// 40 Visualizations/IO_FB/Parameter/Parameter_DO/VIS_PARAMETER_TEMP_DO
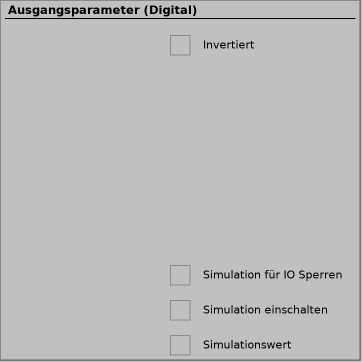
VISUALIZATION VIS_PARAMETER_TEMP_DO  // 362x362
VAR_INPUT
    ITF_DO_IN	:  	ITF_DO;
END_VAR
    RoundedRectangle (0,0 360x360)
    Label (5,0 350x20), "Ausgangsparameter (Digital)"
    Line (5,18) (355,18)
    Frame (170,35 20x20)
        shows CtaSysConfig.visBOOL(visfbBOOLIn := ITF_DO_IN.P_scfbDO_fbxInvert)
    Label (200,35 150x20), "Invertiert"
    Frame (170,335 20x20), invisible if: CtaSysConfig.fcGetEnumerationId(ITF_DO_IN.P_scfbIO_fbxSimulationLock) = 1
        shows CtaSysConfig.visBOOL(visfbBOOLIn := ITF_DO_IN.P_scfbDO_fbxSimulationValue)
    Label (200,335 150x20), "Simulationswert", invisible if: CtaSysConfig.fcGetEnumerationId(ITF_DO_IN.P_scfbIO_fbxSimulationLock) = 1
    Frame (170,265 20x20)
        shows CtaSysConfig.visBOOL(visfbBOOLIn := ITF_DO_IN.P_scfbIO_fbxSimulationLock)
    Label (200,300 150x20), "Simulation einschalten", invisible if: CtaSysConfig.fcGetEnumerationId(ITF_DO_IN.P_scfbIO_fbxSimulationLock) = 1
    Label (200,265 150x20), "Simulation für IO Sperren"
    Frame (170,300 20x20), invisible if: CtaSysConfig.fcGetEnumerationId(ITF_DO_IN.P_scfbIO_fbxSimulationLock) = 1
        shows CtaSysConfig.visBOOL(visfbBOOLIn := ITF_DO_IN.P_scfbIO_Simulation)
END_VISUALIZATION

// 40 Visualizations/IO_FB/DI/SimDI_Temp_Querry
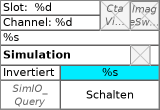
VISUALIZATION SimDI_Temp_Querry  // 160x110
VAR_INPUT
	ITF_DI : ITF_DI;
END_VAR
    Frame (0,0 160x110)
        shows SimDI_Temp(ITF_DI := ITF_DI)
END_VISUALIZATION

// 40 Visualizations/IO_FB/DO/SimDO_Temp_Querry
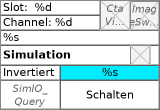
VISUALIZATION SimDO_Temp_Querry  // 160x110
VAR_INPUT	
	ITF_DO : ITF_DO;
END_VAR
    Frame (0,0 160x110)
        shows SimDO_Temp(ITF_DO := ITF_DO)
END_VISUALIZATION

// 40 Visualizations/IO_MANAGER/DEVICE/VIS_DEVICE_QUERY
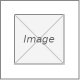
VISUALIZATION VIS_DEVICE_QUERY  // 80x80
VAR_INPUT
	ITF_IO_DEVICE_IN	:	ITF_IO_DEVICE;	
END_VAR
VAR
    fbDialog    	:   VU.FbOpenDialogExtended;
END_VAR
    Image (14,14 50x50), colour toggle: ITF_IO_DEVICE_IN.ERROR, input disabled if: ITF_IO_DEVICE_IN.proVISU_DIA_NAME = ''
        p84334746: ITF_IO_DEVICE_IN.IMAGE
        OnMouseClick: execute {
            ITF_IO_DEVICE_IN.RELOAD_ARRAY(TRUE,FALSE,FALSE);
            fbDialog(itfClientFilter            := VU.Globals.CurrentClient,
                     xExecute                   := FALSE,
            		 xModal						:= FALSE,
                     sDialogName                := ITF_IO_DEVICE_IN.proVISU_DIA_NAME,
                     pbyDialogInterfaceData     := ADR(ITF_IO_DEVICE_IN),
                     udiDialogInterfaceDataSize := SIZEOF(ITF_IO_DEVICE_IN));
            fbDialog(itfClientFilter            := VU.Globals.CurrentClient,
                     xExecute                   := TRUE,
            		 xModal						:= FALSE,
                     sDialogName                := ITF_IO_DEVICE_IN.proVISU_DIA_NAME,
                     pbyDialogInterfaceData     := ADR(ITF_IO_DEVICE_IN),
                     udiDialogInterfaceDataSize := SIZEOF(ITF_IO_DEVICE_IN));
        }
    Textfield (0,0 20x15), "%d", text variable: ITF_IO_DEVICE_IN.DEV_NR
    Textfield (0,65 80x15), "%s", text variable: ITF_IO_DEVICE_IN.proGetBMK
END_VISUALIZATION

// 40 Visualizations/IO_MANAGER/DIA_IO_DEVICES
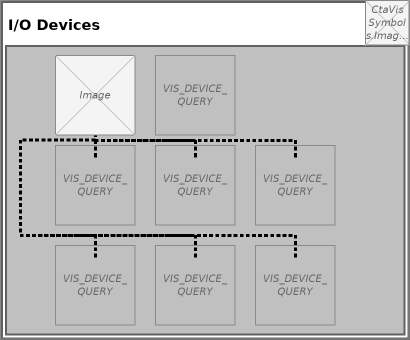
VISUALIZATION DIA_IO_DEVICES  // 410x340
VAR_INPUT
	ITF_IO_MANAGER_IN	:	ITF_IO_MANAGER;	
END_VAR
    RoundedRectangle (0,0 410x340)
    Frame (5,45 400x290), invisible if: NOT __QUERYINTERFACE(ITF_IO_MANAGER_IN,ITF_IO_MANAGER_IN)
        shows VIS_IO_DEVICES(ITF_IO_MANAGER_IN := ITF_IO_MANAGER_IN)
    Image (365,0 45x45), image: CtaVisSymbols.ImagePool.close_solo_black
        OnMouseClick:  Dialog=Current Dialog, Result=None, NumpadKeypadSet=True
    Label (5,5 150x40), "I/O Devices"
    InvisibleInput (5,2 360x40)
END_VISUALIZATION

// 40 Visualizations/IO_MANAGER/NETZWERK/VIS_IO_DEVICES
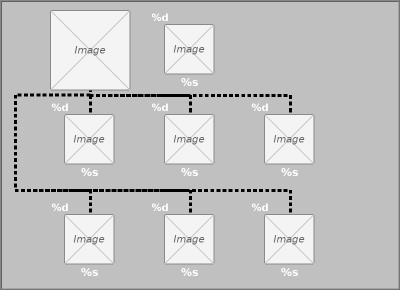
VISUALIZATION VIS_IO_DEVICES  // 400x290
VAR_INPUT
	ITF_IO_MANAGER_IN	:	ITF_IO_MANAGER;	
END_VAR
    Frame (0,0 400x290), invisible if: NOT __QUERYINTERFACE(ITF_IO_MANAGER_IN,ITF_IO_MANAGER_IN)
        shows VIS_IO_DEVICES_NETWORK(ITF_IO_MANAGER_IN := ITF_IO_MANAGER_IN, AY_ITF_DEVICE_VIS := ITF_IO_MANAGER_IN.AY_ITF_DEVICE_VIS)
END_VISUALIZATION

// 40 Visualizations/IO_MANAGER/NETZWERK/VIS_IO_DEVICES_NETWORK
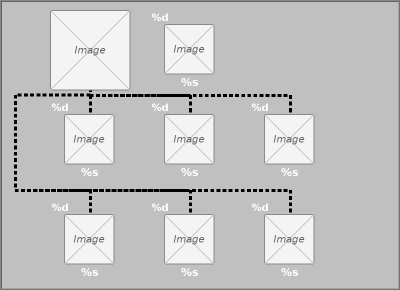
VISUALIZATION VIS_IO_DEVICES_NETWORK  // 400x290
VAR_INPUT
	ITF_IO_MANAGER_IN	:	ITF_IO_MANAGER;	
	AY_ITF_DEVICE_VIS 	: 	ARRAY[0..6] OF ITF_IO_DEVICE;
END_VAR
    RoundedRectangle (0,0 400x290)
    Frame (50,100 80x80)
        shows VIS_DEVICE(ITF_IO_DEVICE_IN := AY_ITF_DEVICE_VIS[1])
    Frame (150,100 80x80)
        shows VIS_DEVICE(ITF_IO_DEVICE_IN := AY_ITF_DEVICE_VIS[2])
    Frame (250,100 80x80)
        shows VIS_DEVICE(ITF_IO_DEVICE_IN := AY_ITF_DEVICE_VIS[3])
    Frame (50,200 80x80)
        shows VIS_DEVICE(ITF_IO_DEVICE_IN := AY_ITF_DEVICE_VIS[4])
    Frame (150,200 80x80)
        shows VIS_DEVICE(ITF_IO_DEVICE_IN := AY_ITF_DEVICE_VIS[5])
    Frame (250,200 80x80)
        shows VIS_DEVICE(ITF_IO_DEVICE_IN := AY_ITF_DEVICE_VIS[6])
    Frame (150,10 80x80)
        shows VIS_DEVICE(ITF_IO_DEVICE_IN := AY_ITF_DEVICE_VIS[0])
    Polyline (90,95) (15,95) (15,190) (90,190) (90,215), invisible if: AY_ITF_DEVICE_VIS[4] = 0
    Polyline (90,95) (15,95) (15,190) (190,190) (190,215), invisible if: AY_ITF_DEVICE_VIS[5] = 0
    Polyline (90,95) (15,95) (15,190) (290,190) (290,215), invisible if: AY_ITF_DEVICE_VIS[6] = 0
    Polyline (90,80) (90,95) (90,95) (290,95) (290,115), invisible if: AY_ITF_DEVICE_VIS[3] = 0
    Polyline (90,80) (90,95) (90,95) (190,95) (190,115), invisible if: AY_ITF_DEVICE_VIS[2] = 0
    Polyline (90,80) (90,95) (90,95) (90,95) (90,115), invisible if: ITF_IO_MANAGER_IN.COUNT = 0 AND AY_ITF_DEVICE_VIS[0] = 0
    Image (50,10 80x80), invisible if: __QUERYINTERFACE(AY_ITF_DEVICE_VIS[0],AY_ITF_DEVICE_VIS[0])
        p84334746: ITF_IO_MANAGER_IN.IMAGE
END_VISUALIZATION

// 40 Visualizations/IO_FB/Simulation/DIA_IO_CONFIG
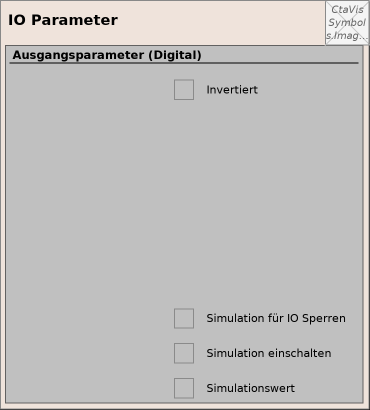
VISUALIZATION DIA_IO_CONFIG  // 370x410
VAR_INPUT
    ITF_IO_IN 	: 	ITF_IO;
END_VAR
    RoundedRectangle (0,0 370x410)
    Frame (5,45 360x360)
        shows VIS_IO_PARAMETER_BASE(ITF_IO_IN := ITF_IO_IN)
    Image (325,0 45x45), image: CtaVisSymbols.ImagePool.close_solo_black
        OnMouseClick:  Dialog=DIA_IO_CONFIG, Result=OK, NumpadKeypadSet=True
    Label (5,5 150x30), "IO Parameter"
    InvisibleInput (5,0 321x45)
END_VISUALIZATION

// 40 Visualizations/IO_TABLE/VIS_IO_TABLE
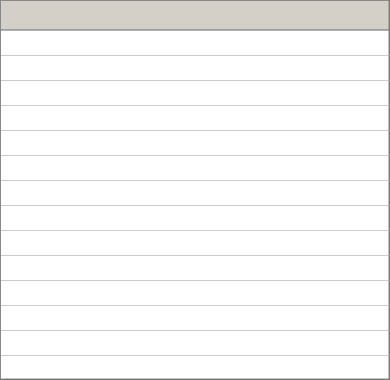
VISUALIZATION VIS_IO_TABLE  // 390x380
VAR_INPUT
	ITF_IO_SLOT_IN	:	ITF_IO_SLOT;	
END_VAR
VAR
	iMax			:	INT;
END_VAR
    Frame (0,0 390x380), invisible if: NOT __QUERYINTERFACE(ITF_IO_SLOT_IN,ITF_IO_SLOT_IN)
        shows VIS_IO_TABLE_QUERY(VIS_IO_TABLE := FC_VIS_IO_TABLE(ITF_IO_SLOT_IN := ITF_IO_SLOT_IN,iMax => iMax), iMax := iMax)
END_VISUALIZATION

// 40 Visualizations/IO_SLOT/VIS_IO_SLOT_IOS_ARRAY
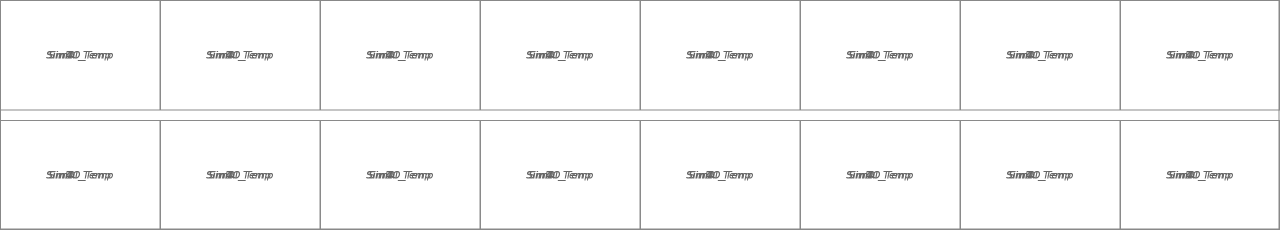
VISUALIZATION VIS_IO_SLOT_IOS_ARRAY  // 1280x230
VAR_INPUT
	AY_ITF_IO_VIS : ARRAY[1..16] OF ITF_IO;	
END_VAR
    Frame (0,0 160x110)
        shows Simulation(ITF_IO := AY_ITF_IO_VIS[1])
    Frame (160,0 160x110)
        shows Simulation(ITF_IO := AY_ITF_IO_VIS[2])
    Frame (320,0 160x110)
        shows Simulation(ITF_IO := AY_ITF_IO_VIS[3])
    Frame (480,0 160x110)
        shows Simulation(ITF_IO := AY_ITF_IO_VIS[4])
    Frame (640,0 160x110)
        shows Simulation(ITF_IO := AY_ITF_IO_VIS[5])
    Frame (800,0 160x110)
        shows Simulation(ITF_IO := AY_ITF_IO_VIS[6])
    Frame (960,0 160x110)
        shows Simulation(ITF_IO := AY_ITF_IO_VIS[7])
    Frame (1120,0 160x110)
        shows Simulation(ITF_IO := AY_ITF_IO_VIS[8])
    Frame (0,120 160x110)
        shows Simulation(ITF_IO := AY_ITF_IO_VIS[9])
    Frame (160,120 160x110)
        shows Simulation(ITF_IO := AY_ITF_IO_VIS[10])
    Frame (320,120 160x110)
        shows Simulation(ITF_IO := AY_ITF_IO_VIS[11])
    Frame (480,120 160x110)
        shows Simulation(ITF_IO := AY_ITF_IO_VIS[12])
    Frame (640,120 160x110)
        shows Simulation(ITF_IO := AY_ITF_IO_VIS[13])
    Frame (800,120 160x110)
        shows Simulation(ITF_IO := AY_ITF_IO_VIS[14])
    Frame (960,120 160x110)
        shows Simulation(ITF_IO := AY_ITF_IO_VIS[15])
    Frame (1120,120 160x110)
        shows Simulation(ITF_IO := AY_ITF_IO_VIS[16])
END_VISUALIZATION

// 40 Visualizations/IO_SLOT/VIS_IO_SLOT_IOS_QUERY
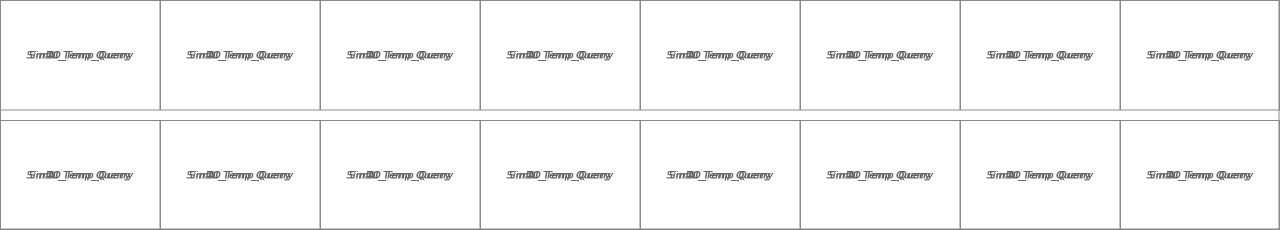
VISUALIZATION VIS_IO_SLOT_IOS_QUERY  // 1280x230
VAR_INPUT
	ITF_IO_SLOT_IN	:	ITF_IO_SLOT;	
END_VAR
    Frame (0,0 1280x230)
        shows VIS_IO_SLOT_IOS_ARRAY(AY_ITF_IO_VIS := ITF_IO_SLOT_IN.AY_ITF_IO_VIS)
END_VISUALIZATION

// 40 Visualizations/IO_SLOT/VIS_IO_SLOT_IOS
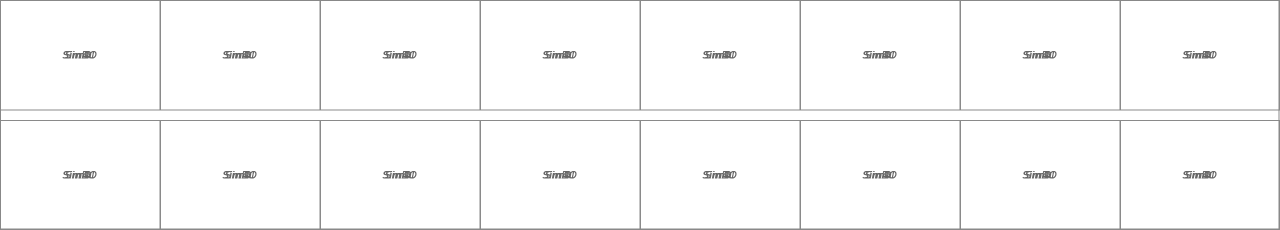
VISUALIZATION VIS_IO_SLOT_IOS  // 1280x230
VAR_INPUT
	ITF_IO_SLOT_IN	:	ITF_IO_SLOT;	
END_VAR
    Frame (0,0 1280x230), invisible if: NOT __QUERYINTERFACE(ITF_IO_SLOT_IN,ITF_IO_SLOT_IN)
        shows VIS_IO_SLOT_IOS_QUERY(ITF_IO_SLOT_IN := ITF_IO_SLOT_IN)
END_VISUALIZATION

// 40 Visualizations/IO_TABLE/VIS_IO_TABLE_QUERY
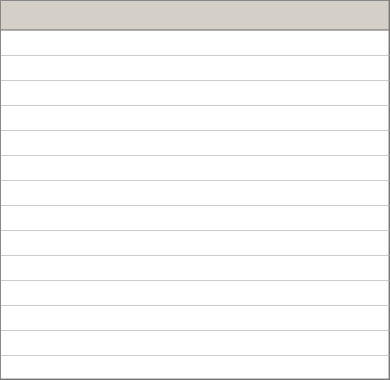
VISUALIZATION VIS_IO_TABLE_QUERY  // 390x380
VAR_INPUT
	VIS_IO_TABLE 	: ARRAY[1..18] OF ITF_IO_TABLE;
	iMax			: INT;
END_VAR
    Table (0,0 390x380), data array: VIS_IO_TABLE
        p1014161805: 18 - 1 + INT#1
        p1128707560: iMax
        p4242324053: FC_VIS_IO_TABLE(ITF_IO_SLOT_IN)[INDEX].proOkVisu
        p1739542657: FC_VIS_IO_TABLE(ITF_IO_SLOT_IN)[INDEX].proOK
        p516019884: FC_VIS_IO_TABLE(ITF_IO_SLOT_IN)[INDEX].proLogName
        p2243050616: FC_VIS_IO_TABLE(ITF_IO_SLOT_IN)[INDEX].proIsSimLocked
        p4088588272: FC_VIS_IO_TABLE(ITF_IO_SLOT_IN)[INDEX].proIsBOOL_IO
        p1757482276: FC_VIS_IO_TABLE(ITF_IO_SLOT_IN)[INDEX].PARENT
        p2192122294: FC_VIS_IO_TABLE(ITF_IO_SLOT_IN)[INDEX].proPhysikalValueVisu
        p400160035: FC_VIS_IO_TABLE(ITF_IO_SLOT_IN)[INDEX].ProSetInstancePathOnDynCreate
        p1265227338: FC_VIS_IO_TABLE(ITF_IO_SLOT_IN)[INDEX].proSimVisu
        p3726181087: FC_VIS_IO_TABLE(ITF_IO_SLOT_IN)[INDEX].SELF
        p3136911649: FC_VIS_IO_TABLE(ITF_IO_SLOT_IN)[INDEX].SELFPOINTER^
        p3854506369: VIS_IO_TABLE[INDEX].IO_NR
        p2170511999: VIS_IO_TABLE[INDEX].proPhysikalValueVisu
        p3723444502: VIS_IO_TABLE[INDEX].proSimVisu
        p1218418051: VIS_IO_TABLE[INDEX].SLOT_NR
        p2232123230: SLOT NR
        p511219082: IO NR
        p1755163831: IO TYPE
        p1791247317: VIS_IO_TABLE[INDEX].IO_TYPE
        p262371475: VIS_IO_TABLE[INDEX].proOkVisu
END_VISUALIZATION

// 40 Visualizations/IO_FB/IO/SimIO
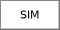
VISUALIZATION SimIO  // 60x30
VAR_INPUT	
	ITF_IO : ITF_IO;
END_VAR
VAR
	ITF_BOOL : CtaSysConfig.ITF_BOOL;
END_VAR
    Frame (0,0 60x30), invisible if: NOT __QUERYINTERFACE(ITF_IO.P_scfbIO_Simulation,ITF_BOOL), input disabled if: ITF_IO.proIsSimLocked
        shows SimIO_Temp(ITF_BOOL := ITF_BOOL)
END_VISUALIZATION

// 40 Visualizations/IO_FB/IO/SimIO_Query
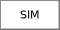
VISUALIZATION SimIO_Query  // 60x30
VAR_INPUT	
	ITF_BOOL : CtaSysConfig.ITF_BOOL;
END_VAR
    RoundedRectangle (0,0 60x30), "SIM", colour toggle: ITF_BOOL.proValue
        toggle ITF_BOOL.proValue
END_VISUALIZATION

// 40 Visualizations/IO_FB/DO/SimValue/SimDO_Value
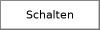
VISUALIZATION SimDO_Value  // 100x30
VAR_INPUT	
	ITF_DO : ITF_DO;
END_VAR
VAR
	ITF_BOOL : CtaSysConfig.ITF_BOOL;
END_VAR
    Frame (0,0 100x30), invisible if: NOT __QUERYINTERFACE(ITF_DO.P_scfbDO_fbxSimulationValue,ITF_BOOL), input disabled if: ITF_DO.proIsSimLocked
        shows SimDO_Value_Query(ITF_DO := ITF_DO, ITF_BOOL := ITF_BOOL)
END_VISUALIZATION

// 40 Visualizations/IO_FB/DO/SimValue/SimDO_Value_Query
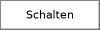
VISUALIZATION SimDO_Value_Query  // 100x30
VAR_INPUT	
	ITF_DO 		: ITF_DO;
	ITF_BOOL 	: CtaSysConfig.ITF_BOOL;
END_VAR
    RoundedRectangle (0,0 100x30), "Schalten", colour toggle: ITF_DO.proValue
        toggle ITF_BOOL.proValue
END_VISUALIZATION

// 40 Visualizations/IO_FB/IO/Invert/SimInvert
VISUALIZATION SimInvert  // 60x15
VAR_INPUT	
	ITF_BOOL : CtaSysConfig.ITF_BOOL;
END_VAR
    Frame (0,0 60x15), invisible if: NOT __QUERYINTERFACE(ITF_BOOL,ITF_BOOL)
        shows SimInvert_Query(ITF_BOOL := ITF_BOOL)
END_VISUALIZATION

// 40 Visualizations/IO_FB/DI/SimValue/SimDI_Value
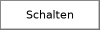
VISUALIZATION SimDI_Value  // 100x30
VAR_INPUT	
	ITF_DI : ITF_DI;
END_VAR
VAR
	ITF_BOOL : CtaSysConfig.ITF_BOOL;
END_VAR
    Frame (0,0 100x30), invisible if: NOT __QUERYINTERFACE(ITF_DI.P_scfbDI_fbxSimulationValue,ITF_BOOL), input disabled if: ITF_DI.proIsSimLocked
        shows SimDI_Value_Query(ITF_DI := ITF_DI, ITF_BOOL := ITF_BOOL)
END_VISUALIZATION

// 40 Visualizations/IO_FB/DI/SimValue/SimDI_Value_Query
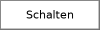
VISUALIZATION SimDI_Value_Query  // 100x30
VAR_INPUT	
	ITF_DI 		: ITF_DI;
	ITF_BOOL 	: CtaSysConfig.ITF_BOOL;
END_VAR
    RoundedRectangle (0,0 100x30), "Schalten", colour toggle: ITF_DI.proValue
        toggle ITF_BOOL.proValue
END_VISUALIZATION

// 40 Visualizations/IO_FB/IO/SimIO_Temp
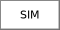
VISUALIZATION SimIO_Temp  // 60x30
VAR_INPUT	
	ITF_BOOL : CtaSysConfig.ITF_BOOL;
END_VAR
    Frame (0,0 60x30), invisible if: NOT __QUERYINTERFACE(ITF_BOOL,ITF_BOOL)
        shows SimIO_Query(ITF_BOOL := ITF_BOOL)
END_VISUALIZATION

// 40 Visualizations/IO_FB/IO/Invert/SimInvert_Query
VISUALIZATION SimInvert_Query  // 60x15
VAR_INPUT	
	ITF_BOOL : CtaSysConfig.ITF_BOOL;
END_VAR
    Rectangle (0,0 60x15), colour toggle: ITF_BOOL.proValue
    Label (0,0 60x15), "Invertiert", invisible if: NOT ITF_BOOL.proValue
END_VISUALIZATION

(* text list txtIOType (id | default)
  Unknown | Unbekannt
  Digital_IN | Digital IN
  Digital_OUT | Digital OUT
  DC_0_10V_OUT | DC 0-10V OUT
  DC_4_20mA_OUT | DC 4-20mA OUT
  DC_0_10V_IN | DC 0-10V IN
  DC_4_20mA_IN | DC 4-20mA IN
  OHM | Ohm
  DC_0_20mA_OUT | DC 0-20mA OUT
  TEMPERATUR | Temperatur
  DC_0_20mA_IN | DC 0-20mA IN
   |  *)

(* text list txtWarning (id | default)
  91 | IO Handeingriff
   |  *)

(* text list txtError (id | default)
  91 | K-Bus Error Reboot notwendig
  92 | Modulkonfigurations Fehler. Module stimmen nicht mit Software überein
   |  *)

(* text list txtPhysicalUnit (id | default)
  0 | NaN
  1 | Digital In
  2 | Digital Out
  3 | 0 - 10 V
  4 | 4 - 20 mA
  5 | 0 - 10 V
  6 | 4 - 20 mA
  7 | Ohm
  8 | 0 - 20 mA
  9 | °C
  10 | 0 - 20 mA
   |  *)
